(* Logix 5000 project; controller Transcat_L33ER vendor 1 type 14 code 107 rev 32.11; software revision 32.02; part 5 of 5 *)
(* tags used below, declared in another part *)
   ActiveRecipe : Recipe;   // Active process recipe downloaded from the HMI recipe system and used by the PLC for automatic operation.
   alwaysOFF : BOOL;
   AnyAutoRun : BOOL;   // Bit that in on if ANY device is placed into Auto run (to signal pre-start beed)
   AnyManualRun : BOOL;   // Bit that in on if ANY device is placed into manual run (to signal pre-start beed)
   BeaconBlueLight : ALIAS FOR TC_Remote_IO:3:O.3;   // Blue Beacon Light
   BeaconGreenLight : ALIAS FOR TC_Remote_IO:3:O.2;   // Green Beacon Light
   BeaconRedLight : ALIAS FOR TC_Remote_IO:3:O.0;   // Red Beacon Light
   BeaconYellowLight : ALIAS FOR TC_Remote_IO:3:O.1;   // Yellow Beacon Light
   Beep : BOOL;   // Bit to Activte Beacon Alarm
   BeepNew : ALIAS FOR TC_Remote_IO:3:O.4;
   Device : Device[20];
   FT103 : BronkhorstFlowMeter;
   FT104 : BronkhorstFlowMeter;
   FT105 : BronkhorstFlowMeter;
   GF101 : Thayer_WB_Feeder;   // Thayer 1 Tags
   GF201 : Thayer_WB_Feeder;   // Thayer 2 Tags
   GF301 : Acrison_Feeder;   // GF103 - Small Feeder 1
   GreenFlashingOff : TIMER;
   GreenFlashingOn : TIMER;
   MSG_FROM_SLC500 : INT[10];
   MX101 : Howes_Mixer;
   MX201 : Howes_Mixer;
   RecipeAnyDeviceSelected : BOOL;   // True when at least one device is selected for automatic operation in the active recipe.
   RecipeParametersValid : BOOL;   // True when all selected devices contain valid recipe operating parameters.
   rNum : DINT;   // Index used by RecipeManager to process active recipe device parameters.
   StartBeepTimer : TIMER;   // Timer to sound the beep alarm before starting a device
   UpperHowesSpeed : INT;
   VF101 : Acrison_Feeder;   // Medium Feeder Tags
   VF201 : Acrison_Feeder;   // Small Feeder 2 Tags
   VFD_Panel_Safety_Hoist_1_Cart_OK : ALIAS FOR XS26_VFD_Cabinet_Safety_Controller:I1.Data[2].2;   // HOIST 1 Cart Sensor
   VFD_Panel_Safety_Hoist_2_Cart_OK : ALIAS FOR XS26_VFD_Cabinet_Safety_Controller:I1.Data[2].3;   // HOIST 2 Cart Sensor
   YellowFlashOff : TIMER;
   YellowFlashOn : TIMER;
(* MainProgram, continued *)

ROUTINE Light_Beacon   (* ladder *)
// Indicator Light Beacon
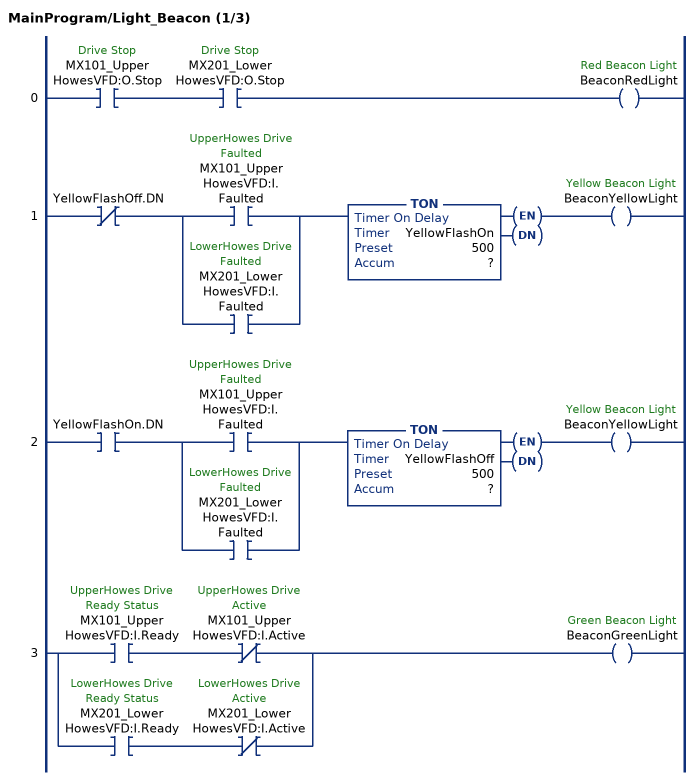
   0: XIC(MX101_UpperHowesVFD:O.Stop)XIC(MX201_LowerHowesVFD:O.Stop)OTE(BeaconRedLight);
   1: XIO(YellowFlashOff.DN)[XIC(MX101_UpperHowesVFD:I.Faulted) ,XIC(MX201_LowerHowesVFD:I.Faulted) ]TON(YellowFlashOn,?,?)OTE(BeaconYellowLight);
   2: XIC(YellowFlashOn.DN)[XIC(MX101_UpperHowesVFD:I.Faulted) ,XIC(MX201_LowerHowesVFD:I.Faulted) ]TON(YellowFlashOff,?,?)OTE(BeaconYellowLight);
   3: [XIC(MX101_UpperHowesVFD:I.Ready) XIO(MX101_UpperHowesVFD:I.Active) ,XIC(MX201_LowerHowesVFD:I.Ready) XIO(MX201_LowerHowesVFD:I.Active) ]OTE(BeaconGreenLight);
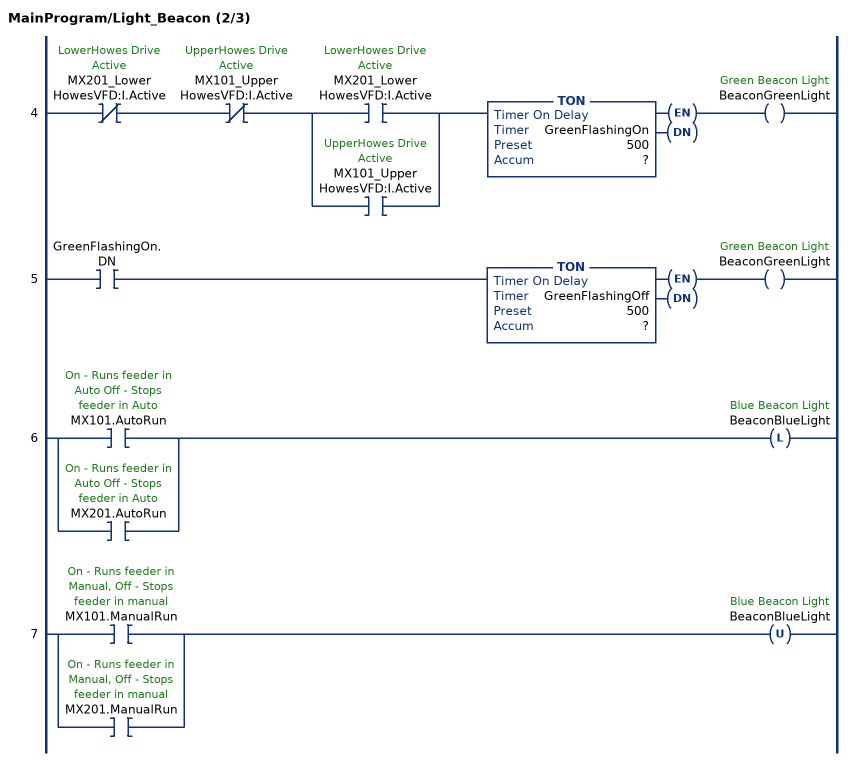
   4: XIO(MX201_LowerHowesVFD:I.Active)XIO(MX101_UpperHowesVFD:I.Active)[XIC(MX201_LowerHowesVFD:I.Active) ,XIC(MX101_UpperHowesVFD:I.Active) ]TON(GreenFlashingOn,?,?)OTE(BeaconGreenLight);
   5: XIC(GreenFlashingOn.DN)TON(GreenFlashingOff,?,?)OTE(BeaconGreenLight);
   6: [XIC(MX101.AutoRun) ,XIC(MX201.AutoRun) ]OTL(BeaconBlueLight);
   7: [XIC(MX101.ManualRun) ,XIC(MX201.ManualRun) ]OTU(BeaconBlueLight);
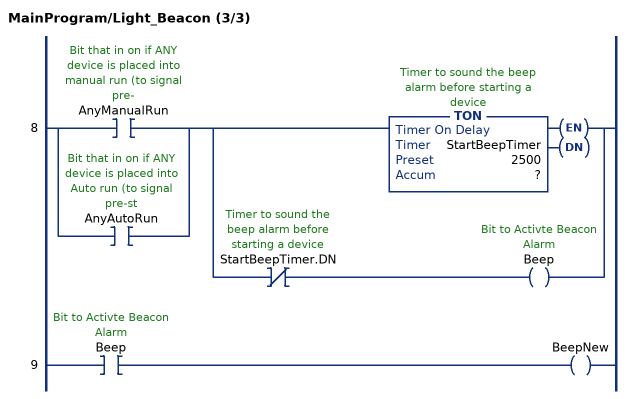
   8: [XIC(AnyManualRun) ,XIC(AnyAutoRun) ][TON(StartBeepTimer,?,?) ,XIO(StartBeepTimer.DN) OTE(Beep) ];
   9: XIC(Beep)OTE(BeepNew);
END_ROUTINE

ROUTINE MainRoutine   (* ladder *)
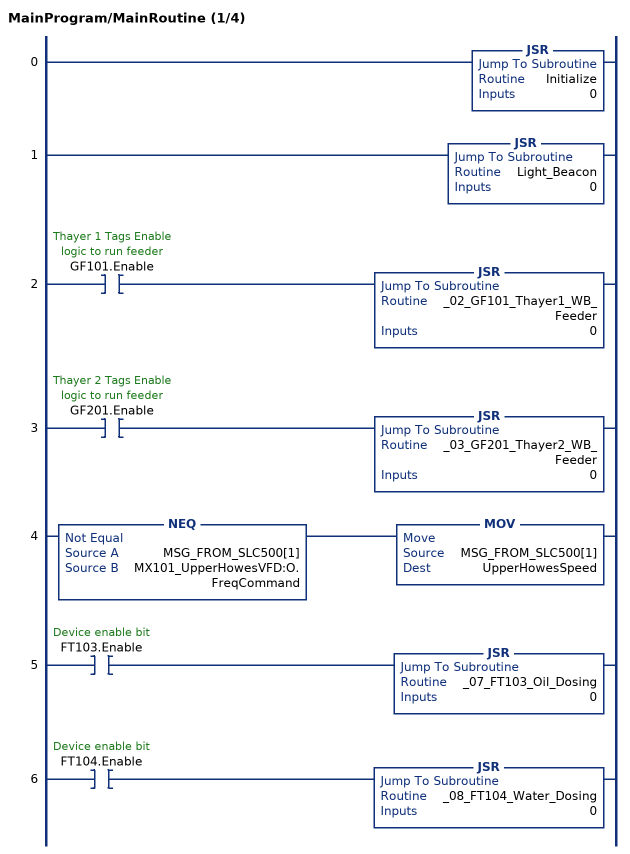
   0: JSR(Initialize,0);
   1: JSR(Light_Beacon,0);
   2: XIC(GF101.Enable)JSR(_02_GF101_Thayer1_WB_Feeder,0);
   3: XIC(GF201.Enable)JSR(_03_GF201_Thayer2_WB_Feeder,0);
   4: NEQ(MSG_FROM_SLC500[1],MX101_UpperHowesVFD:O.FreqCommand)MOV(MSG_FROM_SLC500[1],UpperHowesSpeed);
   5: XIC(FT103.Enable)JSR(_07_FT103_Oil_Dosing,0);
   6: XIC(FT104.Enable)JSR(_08_FT104_Water_Dosing,0);
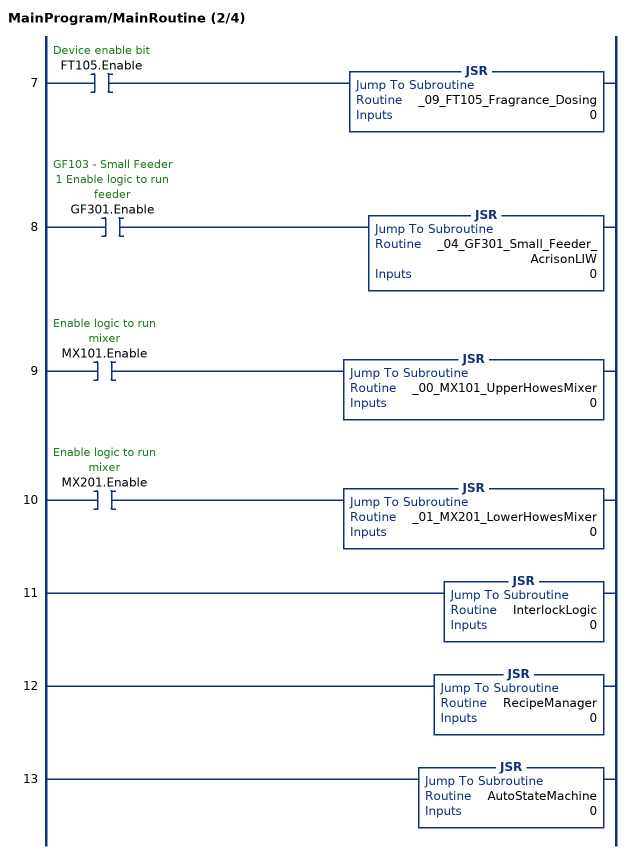
   7: XIC(FT105.Enable)JSR(_09_FT105_Fragrance_Dosing,0);
   8: XIC(GF301.Enable)JSR(_04_GF301_Small_Feeder_AcrisonLIW,0);
   9: XIC(MX101.Enable)JSR(_00_MX101_UpperHowesMixer,0);
   10: XIC(MX201.Enable)JSR(_01_MX201_LowerHowesMixer,0);
   11: JSR(InterlockLogic,0);
   12: JSR(RecipeManager,0);
   13: JSR(AutoStateMachine,0);
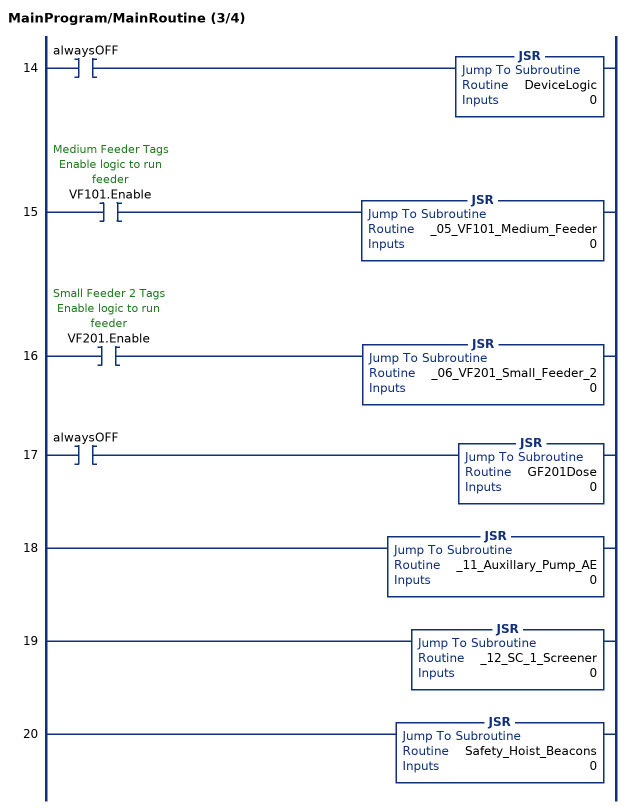
   14: XIC(alwaysOFF)JSR(DeviceLogic,0);
   15: XIC(VF101.Enable)JSR(_05_VF101_Medium_Feeder,0);
   16: XIC(VF201.Enable)JSR(_06_VF201_Small_Feeder_2,0);
   17: XIC(alwaysOFF)JSR(GF201Dose,0);
   18: JSR(_11_Auxillary_Pump_AE,0);
   19: JSR(_12_SC_1_Screener,0);
   20: JSR(Safety_Hoist_Beacons,0);
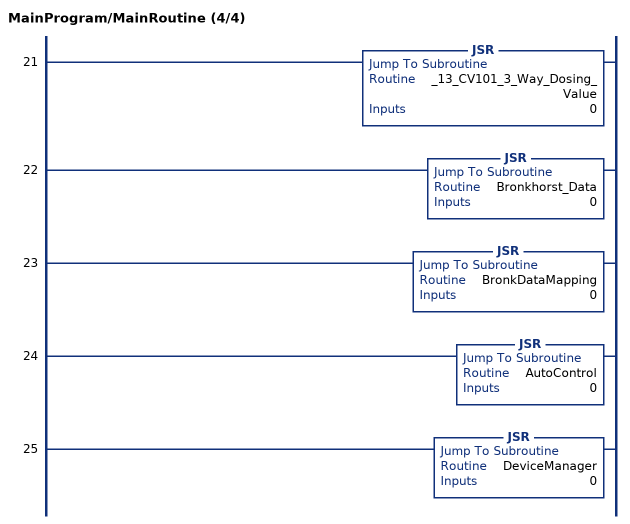
   21: JSR(_13_CV101_3_Way_Dosing_Value,0);
   22: JSR(Bronkhorst_Data,0);
   23: JSR(BronkDataMapping,0);
   24: JSR(AutoControl,0);
   25: JSR(DeviceManager,0);
END_ROUTINE

ROUTINE RecipeDeviceLogic   (* ladder *)
// Processes and validates recipe parameters for each device during the RecipeManager FOR loop.
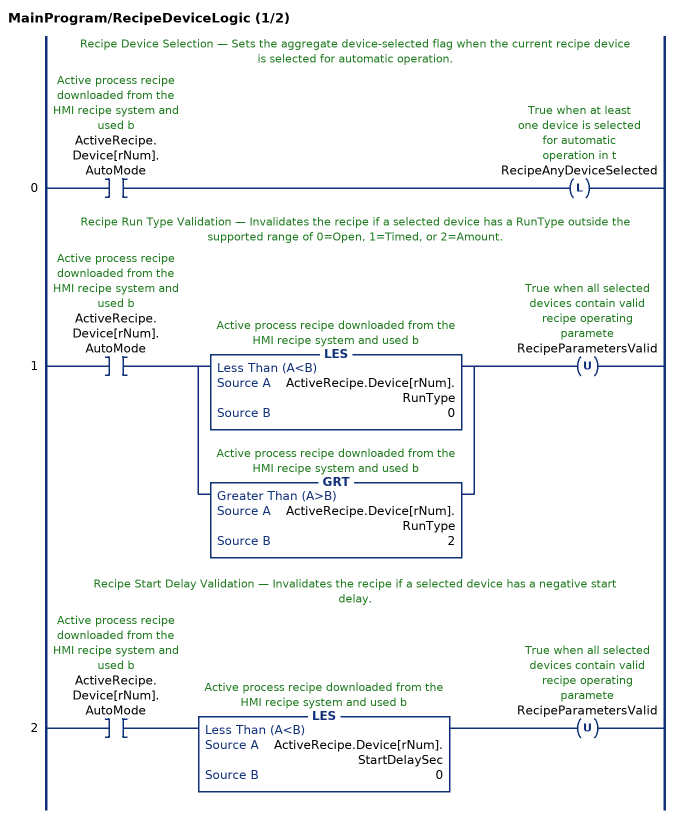
   // Recipe Device Selection — Sets the aggregate device-selected flag when the current recipe device is selected for automatic operation.
   0: XIC(ActiveRecipe.Device[rNum].AutoMode)OTL(RecipeAnyDeviceSelected);
   // Recipe Run Type Validation — Invalidates the recipe if a selected device has a RunType outside the supported range of 0=Open, 1=Timed, or 2=Amount.
   1: XIC(ActiveRecipe.Device[rNum].AutoMode)[LES(ActiveRecipe.Device[rNum].RunType,0) ,GRT(ActiveRecipe.Device[rNum].RunType,2) ]OTU(RecipeParametersValid);
   // Recipe Start Delay Validation — Invalidates the recipe if a selected device has a negative start delay.
   2: XIC(ActiveRecipe.Device[rNum].AutoMode)LES(ActiveRecipe.Device[rNum].StartDelaySec,0)OTU(RecipeParametersValid);
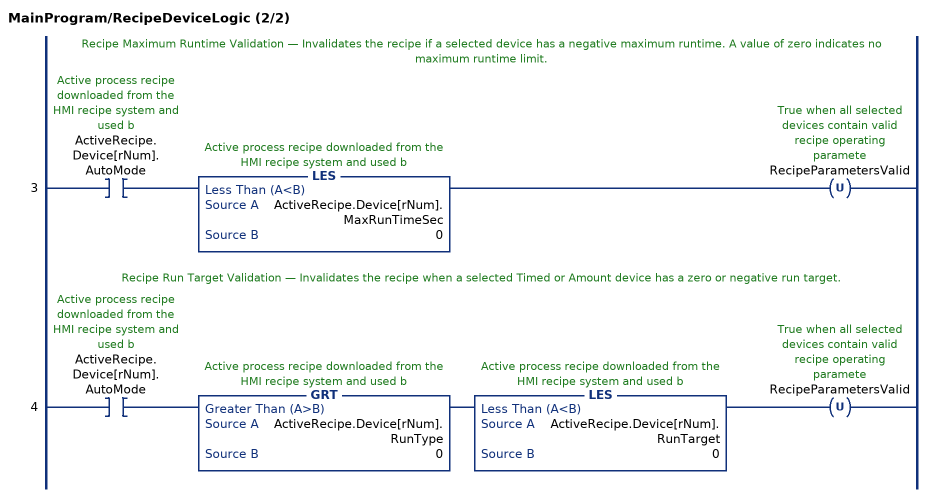
   // Recipe Maximum Runtime Validation — Invalidates the recipe if a selected device has a negative maximum runtime. A value of zero indicates no maximum runtime limit.
   3: XIC(ActiveRecipe.Device[rNum].AutoMode)LES(ActiveRecipe.Device[rNum].MaxRunTimeSec,0)OTU(RecipeParametersValid);
   // Recipe Run Target Validation — Invalidates the recipe when a selected Timed or Amount device has a zero or negative run target.
   4: XIC(ActiveRecipe.Device[rNum].AutoMode)GRT(ActiveRecipe.Device[rNum].RunType,0)LES(ActiveRecipe.Device[rNum].RunTarget,0)OTU(RecipeParametersValid);
END_ROUTINE

ROUTINE RecipeManager   (* ladder *)
// validated and prepares ActiveRecipe
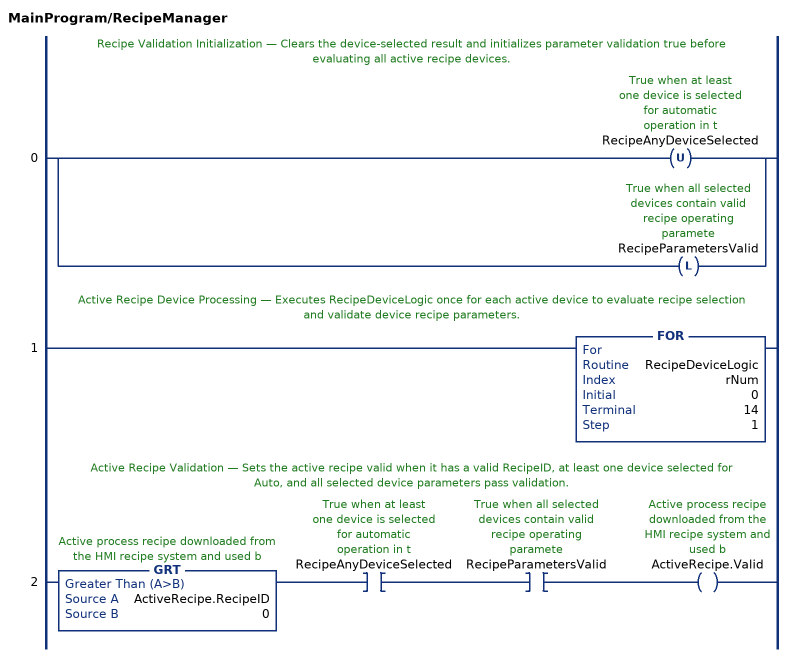
   // Recipe Validation Initialization — Clears the device-selected result and initializes parameter validation true before evaluating all active recipe devices.
   0: [OTU(RecipeAnyDeviceSelected) ,OTL(RecipeParametersValid) ];
   // Active Recipe Device Processing — Executes RecipeDeviceLogic once for each active device to evaluate recipe selection and validate device recipe parameters.
   1: FOR(RecipeDeviceLogic,rNum,0,14,1);
   // Active Recipe Validation — Sets the active recipe valid when it has a valid RecipeID, at least one device selected for Auto, and all selected device parameters pass validation.
   2: GRT(ActiveRecipe.RecipeID,0)XIC(RecipeAnyDeviceSelected)XIC(RecipeParametersValid)OTE(ActiveRecipe.Valid);
END_ROUTINE

ROUTINE Safety_Hoist_Beacons   (* ladder *)
// Saety Hoist Light Beacons
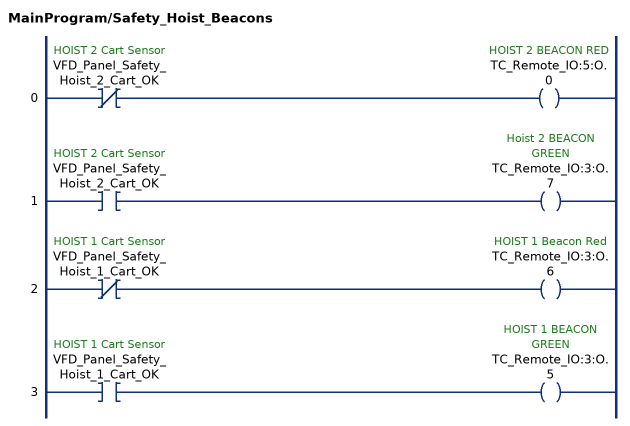
   0: XIO(VFD_Panel_Safety_Hoist_2_Cart_OK)OTE(TC_Remote_IO:5:O.0);
   1: XIC(VFD_Panel_Safety_Hoist_2_Cart_OK)OTE(TC_Remote_IO:3:O.7);
   2: XIO(VFD_Panel_Safety_Hoist_1_Cart_OK)OTE(TC_Remote_IO:3:O.6);
   3: XIC(VFD_Panel_Safety_Hoist_1_Cart_OK)OTE(TC_Remote_IO:3:O.5);
END_ROUTINE
END_PROGRAM
